// TIA Portal V15.1 export
// export: Created 2026-01-15T16:29:49.2237765Z, ExportSetting WithDefaults, WithReadOnly, DisplayName Totally Integrated Automation Portal, DisplayVersion V15.1 Update 8, DisplayName TIA Portal Openness, DisplayVersion V15.1 Update 8, DisplayName STEP 7 Professional, DisplayVersion V15.1 Update 8, DisplayName WinCC Advanced, DisplayVersion V15.1 Update 8
VAR_GLOBAL   // PLC tag table "Default tag table_1"
   System_Byte AT %MB1 : Byte;
   FirstScan AT %M1.0 : Bool;
   DiagStatusUpdate AT %M1.1 : Bool;
   AlwaysTRUE AT %M1.2 : Bool;
   AlwaysFALSE AT %M1.3 : Bool;
   Clock_Byte AT %MB0 : Byte;
   Clock_10Hz AT %M0.0 : Bool;
   Clock_5Hz AT %M0.1 : Bool;
   "Clock_2.5Hz" AT %M0.2 : Bool;
   Clock_2Hz AT %M0.3 : Bool;
   "Clock_1.25Hz" AT %M0.4 : Bool;
   Clock_1Hz AT %M0.5 : Bool;
   "Clock_0.625Hz" AT %M0.6 : Bool;
   "Clock_0.5Hz" AT %M0.7 : Bool;
   "NAP LIEU" AT %M200.0 : Bool;
   "RUA NOI" AT %M200.1 : Bool;
   TH_NAP_WAG AT %M300.0 : Bool;
   TH_NAP_WAP AT %M300.2 : Bool;
   TH_NAP_WFD AT %M300.1 : Bool;
   TH_NAP_WSB AT %M300.3 : Bool;
   "LUU_CAN TAY" AT %M200.2 : Bool;
   "LUU TAY CEM1" AT %M200.3 : Bool;
   "LUU TAY CEM2" AT %M200.4 : Bool;
   "LUU TAY WAT1" AT %M200.5 : Bool;
   "LUU TAY ADD1" AT %M200.6 : Bool;
   XA_HET_AGG AT %M200.7 : Bool;
   "LUU TAY WAG1" AT %M210.0 : Bool;
   "LUU TAY WAG2" AT %M210.1 : Bool;
   "LUU TAY WAG3" AT %M210.2 : Bool;
   "LUU TAY WAG4" AT %M210.3 : Bool;
   "LUU TAY WAG5" AT %M210.4 : Bool;
END_VAR
VAR_GLOBAL CONSTANT   // user constants
   "Local(1)" : Hw_SubModule := 50;
   "Local~PROFINET_interface_1(1)" : Hw_Interface := 64;
   "Local~PROFINET_interface_1~Port_1(1)" : Hw_Interface := 65;
   "Local~HSC_1(1)" : Hw_Hsc := 257;
   "Local~HSC_2(1)" : Hw_Hsc := 258;
   "Local~HSC_3(1)" : Hw_Hsc := 259;
   "Local~HSC_4(1)" : Hw_Hsc := 260;
   "Local~HSC_5(1)" : Hw_Hsc := 261;
   "Local~HSC_6(1)" : Hw_Hsc := 262;
   "Local~AI_2_1(1)" : Hw_SubModule := 263;
   "Local~DI_14_DQ_10_1(1)" : Hw_SubModule := 264;
   "Local~Pulse_1(1)" : Hw_Pwm := 265;
   "Local~Pulse_2(1)" : Hw_Pwm := 266;
   "OB_Main_P1(1)" : OB_PCYCLE := 1;
   "Local~Pulse_3(1)" : Hw_Pwm := 267;
   "Local~Pulse_4(1)" : Hw_Pwm := 268;
   "None(1)" : Pip := 65535;
   "Automatic update(1)" : Pip := 0;
   "PIP 1(1)" : Pip := 1;
   "PIP 2(1)" : Pip := 2;
   "PIP 3(1)" : Pip := 3;
   "PIP 4(1)" : Pip := 4;
   "PIP OB Servo(1)" : Pip := 32768;
   "Local~DQ_8xRelay_1(1)" : Hw_SubModule := 273;
   "Local~AI_4x13BIT_1(1)" : Hw_SubModule := 271;
   "Local~AI_4xTC_1(1)" : Hw_SubModule := 272;
   "Local~DI_8_DQ_8x24VDC_1" : Hw_SubModule := 274;
   "Local~DQ_16xRelay_1(1)" : Hw_SubModule := 269;
   "Local~AI_4x13BIT_2(1)" : Hw_SubModule := 270;
END_VAR
